Omron Sysmac Studio project UAMotionLinkLib (Sysmac Studio 1.63.0.7, LibraryProject)
(* For development of UAMotionLinkLib. *)

# Controller LIB: NX102-9000 version 1.64
Axis MC_Axis1, settings changed from default: AxisType=ServoType, FunctionLimit=SingleAxisPTP, UnitsConversion=EnumElement2, UnitsNumerator=8388608, UnitsDenominator=10, TravelDistancePerWorkRotation=5, MaxVelocity=200, MaxJogVelocity=200, InPositionBand=1, ZeroPositionBand=1, FollowingErrorLimit=5, FollowingErrorAlarmLimit=1, EncoderTypes=Abs
Axis MC_Axis2, settings changed from default: AxisNumber=1, AxisType=ServoType, FunctionLimit=SingleAxisPTP, UnitsConversion=EnumElement5, UnitsNumerator=8388608, UnitsDenominator=360, MaxVelocity=36000, MaxJogVelocity=36000, InPositionBand=0.1, ModuloMAXPosition=360, ModuloMINPosition=0
Task PrimaryTask (priority 4, period or condition 2000): ModelTest, ModelTestSimDriveReflection



PROGRAM README
RETURN;
(*

# About This Project
This project is for the development of UAMotionLinkLib.
UAMotionLinkLib provide a model FBs that control a servo via motion FBs published on an OPC UA server.
Currently, UAMotionLinkLib is intended for minor positioning operations such as trial runs and adjustments.

The model FBs are limited to providing wrappers for motion FBs related to positioning.
Servo operation preparation, stop, and emergency stop operations are provided appropriately in the user software,
and it is assumed that these are operating at an appropriate level when using UAMotionLinkLib.


# このプロジェクトについて
このプロジェクトは、UAMotionLinkLibの開発用プロジェクトです。
UAMotionLinkLibは、OPC UAサーバで公開するモーションFBを介してサーボを操作するモデルFBを提供します。
現在、UAMotionLinkLibは、試運転や調整の軽微な位置決め操作を対象としています。

モデルFBは、位置決めに関連したモーションFBのラッパー提供に限ります。
サーボ動作準備、停止、非常停止操作はユーザーソフトウェアにおいて適切に提供され、
UAMotionLinkLib使用時は、それらが適切な水準で動作していることを前提にしています。


For the parts to which I have rights, I follow POU/PROGRAM/LICENSE.
You are free to use and modify it, but we are not responsible for any damage or loss related to it.
*)
END_PROGRAM

PROGRAM LICENSE
RETURN;
(*
The MIT License (MIT)

Copyright(c) 2025 KITA Munemitsu

Permission is hereby granted, free of charge, to any person obtaining a copy of this software and associated
documentation files (the “Software”), to deal in the Software without restriction, including without limitation
the rights to use, copy, modify, merge, publish, distribute, sublicense, and/or sell copies of the Software,
and to permit persons to whom the Software is furnished to do so, subject to the following conditions:

The above copyright notice and this permission notice shall be included in all copies or substantial portions of the Software.

THE SOFTWARE IS PROVIDED “AS IS”, WITHOUT WARRANTY OF ANY KIND, EXPRESS OR IMPLIED, INCLUDING BUT NOT
LIMITED TO THE WARRANTIES OF MERCHANTABILITY, FITNESS FOR A PARTICULAR PURPOSE AND NONINFRINGEMENT.
IN NO EVENT SHALL THE AUTHORS OR COPYRIGHT HOLDERS BE LIABLE FOR ANY CLAIM, DAMAGES OR OTHER LIABILITY,
WHETHER IN AN ACTION OF CONTRACT, TORT OR OTHERWISE, ARISING FROM, OUT OF OR IN CONNECTION WITH THE SOFTWARE
OR THE USE OR OTHER DEALINGS IN THE SOFTWARE.
*)
END_PROGRAM

PROGRAM ModelTest
VAR
    BasicMCController : ModelTest_BasicMCControllerModel;
END_VAR
(*
# About This POU
This is the teesting the information model of UAMotionLinkLib.
Set up an OPC UA server and test that it can be operated by a repository client.

## Usage Steps
1. Prepare Pester for use
   Refer to the following for setup.

   "Installation and Update", Pester, https://pester.dev/docs/introduction/installation

2. Configure the Simulator's OPC UA Server
   Refer to the following for configuring the OPC UA server.

   "OPC UA User's Manual", OMRON Corporation, https://www.fa.omron.co.jp/data_pdf/mnu/w588-e1-15_nj501_nx.pdf?id=3705
   "PwshOpcUaClient", https://github.com/kmu2030/PwshOpcUaClient

   The user and password to register on the OPC UA server are as follows:

   Username: taker
   Password: chocolatepancakes

3. Run the test
   Run the following in the root directory of the cloned repository:

   ```powershell
   Invoke-Pester
   ```


# このPOUについて
UAMotionLinkLibの情報モデルのテスト。
OPC UAサーバを設定し、リポジトリのクライアントで操作できることをテストする。

## 使用手順
1. Pesterを使える状態にする
   以下を参考にセットアップする。
  
  "Installation and Update", Pester, https://pester.dev/docs/introduction/installation

2. シミュレータのOPC UAサーバを設定
   以下を参考にOPC UAサーバを設定する。
  
   "OPC UA User's Manual", OMRON Corporation, https://www.fa.omron.co.jp/data_pdf/mnu/w588-e1-15_nj501_nx.pdf?id=3705
   "PwshOpcUaClient", https://github.com/kmu2030/PwshOpcUaClient

   OPC UAサーバに登録するユーザーとパスワードは以下。

   Username: taker
   Password: chocolatepancakes

3. テストを実行
   以下をリポジトリのクローンのルートディレクトリで実行する。
  
   ```powershell
   Invoke-Pester
   ```

(c) 2025 KITA Munemitsu

*)

IF P_First_Run THEN
	BasicMCController.Enable := TRUE;
END_IF;

BasicMCController();
END_PROGRAM

PROGRAM ModelTestSimDriveReflection
VAR
    iSimMCRefrectors : ARRAY[0..15] OF SimMCReflector;
    i : UINT;
END_VAR
VAR_EXTERNAL CONSTANT
    _MC_AX : ARRAY[0..15] OF _sAXIS_REF;
END_VAR
(*

Reflects the axis command value to the current value when testing the information model of UAMotionLinkLib.


UAMotionLinkLibの情報モデルのテスト時に軸指令値を現在値に反映する。

(c) 2025 KITA Munemitsu

*)

FOR i := 0 TO 15 DO
	iSimMCRefrectors[i](Enable:=TRUE,
						Axis:=_MC_AX[i]);
END_FOR;
END_PROGRAM

FUNCTION_BLOCK BasicMCControllerModel
(* Model FB that provides motion control. *)
VAR
    MoveAbsolute : BasicMCControllerModel_moveAbsolute;
    MoveRelative : BasicMCControllerModel_moveRelative;
    MoveZeroPosition : BasicMCControllerModel_moveZeroPosition;
    Home : BasicMCControllerModel_home;
    SetPosition : BasicMCControllerModel_setPosition;
    Reset : BasicMCControllerModel_reset;
    SetAxisIndex : BasicMCControllerModel_setAxisIndex;
    AxisIndex : UINT := 0;
    Axis : _sAXIS_REF;
END_VAR
VAR_INPUT
    Enable : BOOL;
END_VAR
VAR_IN_OUT CONSTANT
    Axes : ARRAY[*] OF _sAXIS_REF;
END_VAR
VAR_INPUT
    AllowControl : BOOL := False;
END_VAR
VAR_OUTPUT
    Busy : BOOL;
END_VAR
(*

Model FB that provides motion control.


モーション操作を提供するモデルFB。

(c) 2025 KITA Munemitsu

*)

IF Enable <> Busy OR NOT AllowControl THEN
	MoveAbsolute.Execute := FALSE;
	MoveRelative.Execute := FALSE;
	MoveZeroPosition.Execute := FALSE;
	Home.Execute := FALSE;
	SetPosition.Execute := FALSE;
	Reset.Execute := FALSE;
	SetAxisIndex.Execute := FALSE;
	AxisIndex := 0;
END_IF;

Axis := Axes[AxisIndex];

MoveAbsolute(Axis:=Axes[AxisIndex]);
MoveRelative(Axis:=Axes[AxisIndex]);
MoveZeroPosition(Axis:=Axes[AxisIndex]);
Home(Axis:=Axes[AxisIndex]);
SetPosition(Axis:=Axes[AxisIndex]);
Reset(Axis:=Axes[AxisIndex]);
SetAxisIndex(Axes:=Axes, AxisIndex:=AxisIndex);

Busy := Enable
	OR MoveAbsolute.Busy
	OR MoveRelative.Busy
	OR MoveZeroPosition.Busy
	OR Home.Busy
	OR SetPosition.Busy
	OR Reset.Busy;
	
END_FUNCTION_BLOCK

FUNCTION_BLOCK BasicMCControllerModel_setAxisIndex
(* Method FB that specifies the axis to be operated. / This FB is for BasicMCController only. *)
VAR_INPUT
    Execute : BOOL;
END_VAR
VAR_IN_OUT CONSTANT
    Axes : ARRAY[*] OF _sAXIS_REF;
END_VAR
VAR_IN_OUT
    AxisIndex : UINT;
END_VAR
VAR_INPUT
    NewValue : UINT := 0;
END_VAR
VAR_OUTPUT
    Ok : BOOL;
    Done : BOOL;
END_VAR
(*

Method FB that specifies the axis to be operated.
This FB is for BasicMCController only.


操作対象とする軸を指定するメソッドFB。
このFBは、BasicMCController専用。

(c) 2025 KITA Munemitsu

*)

IF NOT Execute THEN
	IF Done THEN
		Ok := FALSE;
		Done := FALSE;
	END_IF;
	
	RETURN;
END_IF;

IF Execute AND NOT Done THEN
	Ok := NewValue < SizeOfAry(Axes);
	IF Ok THEN 
		AxisIndex := NewValue;
	END_IF;
	
	Done := TRUE;
END_IF;
END_FUNCTION_BLOCK

FUNCTION_BLOCK BasicMCControllerModel_moveAbsolute
(* Method FB that is a wrapper for MC_MoveAbsolute. / This FB is for BasicMCController only. *)
VAR
    iMC_MoveAbsolute : MC_MoveAbsolute;
    iState : UINT := 1001;
    iDirection : _eMC_DIRECTION;
    iBufferMode : _eMC_BUFFER_MODE;
END_VAR
VAR_IN_OUT CONSTANT
    Axis : _sAXIS_REF;
END_VAR
VAR_INPUT
    Position : LREAL := 0.0;
    Velocity : LREAL := 0.0;
    Acceleration : LREAL := 0.0;
    Deceleration : LREAL := 0.0;
    Jerk : LREAL := 0.0;
    Direction : UDINT := 0;
    BufferMode : UDINT := 0;
END_VAR
VAR_OUTPUT
    Busy : BOOL;
    Active : BOOL;
    Done : BOOL;
    CommandAborted : BOOL;
    Error : BOOL;
    ErrorID : WORD;
END_VAR
VAR_INPUT
    Execute : BOOL;
END_VAR
(*

Method FB that is a wrapper for MC_MoveAbsolute.
This FB is for BasicMCController only.


MC_MoveAbsoluteのラッパーであるメソッドFB。
このFBは、BasicMCController専用。

(c) 2025 KITA Munemitsu

*)

IF NOT Execute THEN
	IF iState > 0 THEN
		Error := FALSE;
		ErrorID := 0;
		CommandAborted := FALSE;
		Active := FALSE;
		Busy := FALSE;
		Done := FALSE;
		iState := 1001;
		iMC_MoveAbsolute.Execute := FALSE;
	END_IF;
ELSIF Execute AND NOT (Busy OR Done) THEN
	iState := 0;
END_IF;

CASE iState OF
	0:
		iMC_MoveAbsolute.Acceleration := Acceleration;
		iMC_MoveAbsolute.Deceleration := Deceleration;
		iMC_MoveAbsolute.Jerk := Jerk;
		iMC_MoveAbsolute.Position := Position;
		iMC_MoveAbsolute.Velocity := Velocity;
		NumToEnum(In:=Direction, InOut:=iDirection);
		iMC_MoveAbsolute.Direction := iDirection;
		NumToEnum(In:=BufferMode, InOut:=iBufferMode);
		iMC_MoveAbsolute.BufferMode := iBufferMode;
		iMC_MoveAbsolute.Execute := TRUE;
		
		Inc(iState);
	1:
		IF iMC_MoveAbsolute.Done
			OR iMC_MoveAbsolute.Error
			OR iMC_MoveAbsolute.CommandAborted
		THEN
			iMC_MoveAbsolute.Execute := FALSE;
			IF iMC_MoveAbsolute.Error THEN
				Error := TRUE;
				ErrorID := iMC_MoveAbsolute.ErrorID;
			END_IF;
			CommandAborted := iMC_MoveAbsolute.CommandAborted;
			
			Inc(iState);
		END_IF;
	2:
		IF NOT iMC_MoveAbsolute.Busy THEN
			iState := 1000;
		END_IF;
	1000:
		Done := TRUE;

		Inc(iState);
END_CASE;
Busy := iState < 1001;

iMC_MoveAbsolute(Axis:=Axis);
Active := iMC_MoveAbsolute.Active;
END_FUNCTION_BLOCK

FUNCTION_BLOCK BasicMCControllerModel_moveRelative
(* Method FB that is a wrapper for MC_MoveRelative. / This FB is for BasicMCController only. *)
VAR
    iMC_MoveRelative : MC_MoveRelative;
    iState : UINT := 1001;
    iBufferMode : _eMC_BUFFER_MODE;
END_VAR
VAR_INPUT
    Execute : BOOL;
END_VAR
VAR_IN_OUT CONSTANT
    Axis : _sAXIS_REF;
END_VAR
VAR_INPUT
    Distance : LREAL := 0.0;
    Velocity : LREAL := 0.0;
    Acceleration : LREAL := 0.0;
    Deceleration : LREAL := 0.0;
    Jerk : LREAL := 0.0;
    BufferMode : UDINT := 0;
END_VAR
VAR_OUTPUT
    Busy : BOOL;
    Active : BOOL;
    Done : BOOL;
    CommandAborted : BOOL;
    Error : BOOL;
    ErrorID : WORD;
END_VAR
(*

Method FB that is a wrapper for MC_MoveRelative.
This FB is for BasicMCController only.


MC_MoveRelativeのラッパーであるメソッドFB。
このFBは、BasicMCController専用。

(c) 2025 KITA Munemitsu

*)

IF NOT Execute THEN
	IF iState > 0 THEN
		Error := FALSE;
		ErrorID := 0;
		CommandAborted := FALSE;
		Active := FALSE;
		Busy := FALSE;
		Done := FALSE;
		iState := 1001;
		iMC_MoveRelative.Execute := FALSE;
	END_IF;
ELSIF Execute AND NOT (Busy OR Done) THEN
	iState := 0;
END_IF;

CASE iState OF
	0:
		iMC_MoveRelative.Acceleration := Acceleration;
		iMC_MoveRelative.Deceleration := Deceleration;
		iMC_MoveRelative.Jerk := Jerk;
		iMC_MoveRelative.Distance := Distance;
		iMC_MoveRelative.Velocity := Velocity;
		NumToEnum(In:=BufferMode, InOut:=iBufferMode);
		iMC_MoveRelative.BufferMode := iBufferMode;
		iMC_MoveRelative.Execute := TRUE;
		
		Inc(iState);
	1:
		IF iMC_MoveRelative.Done
			OR iMC_MoveRelative.Error
			OR iMC_MoveRelative.CommandAborted
		THEN
			iMC_MoveRelative.Execute := FALSE;
			IF iMC_MoveRelative.Error THEN
				Error := TRUE;
				ErrorID := iMC_MoveRelative.ErrorID;
			END_IF;
			CommandAborted := iMC_MoveRelative.CommandAborted;
			
			Inc(iState);
		END_IF;
	2:
		IF NOT iMC_MoveRelative.Busy THEN
			iState := 1000;
		END_IF;
	1000:
		Done := TRUE;

		Inc(iState);
END_CASE;
Busy := iState < 1001;

iMC_MoveRelative(Axis:=Axis);
Active := iMC_MoveRelative.Active;
END_FUNCTION_BLOCK

FUNCTION_BLOCK BasicMCControllerModel_moveZeroPosition
(* Method FB that is a wrapper for MC_MoveZeroPosition. / This FB is for BasicMCController only. *)
VAR
    iMC_MoveZeroPosition : MC_MoveZeroPosition;
    iState : UINT := 1001;
    iBufferMode : _eMC_BUFFER_MODE;
END_VAR
VAR_INPUT
    Execute : BOOL;
END_VAR
VAR_IN_OUT CONSTANT
    Axis : _sAXIS_REF;
END_VAR
VAR_INPUT
    Velocity : LREAL := 0.0;
    Acceleration : LREAL := 0.0;
    Deceleration : LREAL := 0.0;
    Jerk : LREAL := 0.0;
    BufferMode : UDINT := 0;
END_VAR
VAR_OUTPUT
    Busy : BOOL;
    Active : BOOL;
    Done : BOOL;
    CommandAborted : BOOL;
    Error : BOOL;
    ErrorID : WORD;
END_VAR
(*

Method FB that is a wrapper for MC_MoveZeroPosition.
This FB is for BasicMCController only.


MC_MoveZeroPositionのラッパーであるメソッドFB。
このFBは、BasicMCController専用。

(c) 2025 KITA Munemitsu

*)

IF NOT Execute THEN
	IF iState > 0 THEN
		Error := FALSE;
		ErrorID := 0;
		CommandAborted := FALSE;
		Active := FALSE;
		Busy := FALSE;
		Done := FALSE;
		iState := 1001;
		iMC_MoveZeroPosition.Execute := FALSE;
	END_IF;
ELSIF Execute AND NOT (Busy OR Done) THEN
	iState := 0;
END_IF;

CASE iState OF
	0:
		iMC_MoveZeroPosition.Acceleration := Acceleration;
		iMC_MoveZeroPosition.Deceleration := Deceleration;
		iMC_MoveZeroPosition.Jerk := Jerk;
		iMC_MoveZeroPosition.Velocity := Velocity;
		NumToEnum(In:=BufferMode, InOut:=iBufferMode);
		iMC_MoveZeroPosition.BufferMode := iBufferMode;
		iMC_MoveZeroPosition.Execute := TRUE;
		
		Inc(iState);
	1:
		IF iMC_MoveZeroPosition.Done
			OR iMC_MoveZeroPosition.Error
			OR iMC_MoveZeroPosition.CommandAborted
		THEN
			iMC_MoveZeroPosition.Execute := FALSE;
			IF iMC_MoveZeroPosition.Error THEN
				Error := TRUE;
				ErrorID := iMC_MoveZeroPosition.ErrorID;
			END_IF;
			CommandAborted := iMC_MoveZeroPosition.CommandAborted;
			
			Inc(iState);
		END_IF;
	2:
		IF NOT iMC_MoveZeroPosition.Busy THEN
			iState := 1000;
		END_IF;
	1000:
		Done := TRUE;

		Inc(iState);
END_CASE;
Busy := iState < 1001;

iMC_MoveZeroPosition(Axis:=Axis);
Active := iMC_MoveZeroPosition.Active;
END_FUNCTION_BLOCK

FUNCTION_BLOCK BasicMCControllerModel_home
(* Method FB that is a wrapper for MC_Home. / This FB is for BasicMCController only. *)
VAR
    iMC_Home : MC_Home;
    iState : UINT := 1001;
END_VAR
VAR_INPUT
    Execute : BOOL;
END_VAR
VAR_IN_OUT CONSTANT
    Axis : _sAXIS_REF;
END_VAR
VAR_OUTPUT
    Busy : BOOL;
    Done : BOOL;
    CommandAborted : BOOL;
    Error : BOOL;
    ErrorID : WORD;
END_VAR
(*

Method FB that is a wrapper for MC_Home.
This FB is for BasicMCController only.


MC_HomeのラッパーであるメソッドFB。
このFBは、BasicMCController専用。

(c) 2025 KITA Munemitsu

*)

IF NOT Execute THEN
	IF iState > 0 THEN
		Error := FALSE;
		ErrorID := 0;
		CommandAborted := FALSE;
		Busy := FALSE;
		Done := FALSE;
		iState := 1001;
		iMC_Home.Execute := FALSE;
	END_IF;
ELSIF Execute AND NOT (Busy OR Done) THEN
	iState := 0;
END_IF;

CASE iState OF
	0:
		iMC_Home.Execute := TRUE;
		
		Inc(iState);
	1:
		IF iMC_Home.Done
			OR iMC_Home.Error
			OR iMC_Home.CommandAborted
		THEN
			iMC_Home.Execute := FALSE;
			IF iMC_Home.Error THEN
				Error := TRUE;
				ErrorID := iMC_Home.ErrorID;
			END_IF;
			CommandAborted := iMC_Home.CommandAborted;
			
			Inc(iState);
		END_IF;
	2:
		IF NOT iMC_Home.Busy THEN
			iState := 1000;
		END_IF;
	1000:
		Done := TRUE;

		Inc(iState);
END_CASE;
Busy := iState < 1001;

iMC_Home(Axis:=Axis);
END_FUNCTION_BLOCK

FUNCTION_BLOCK BasicMCControllerModel_setPosition
(* Method FB that is a wrapper for MC_SetPosition. / This FB is for BasicMCController only. *)
VAR
    iMC_SetPosition : MC_SetPosition;
    iState : UINT := 1001;
    iReferenceType : _eMC_REFERENCE_TYPE;
END_VAR
VAR_INPUT
    Execute : BOOL;
END_VAR
VAR_IN_OUT CONSTANT
    Axis : _sAXIS_REF;
END_VAR
VAR_INPUT
    Position : LREAL;
    ReferenceType : UDINT;
END_VAR
VAR_OUTPUT
    Busy : BOOL;
    Done : BOOL;
    CommandAborted : BOOL;
    Error : BOOL;
    ErrorID : WORD;
END_VAR
(*

Method FB that is a wrapper for MC_SetPosition.
This FB is for BasicMCController only.


MC_SetPositionのラッパーであるメソッドFB。
このFBは、BasicMCController専用。

(c) 2025 KITA Munemitsu

*)

IF NOT Execute THEN
	IF iState > 0 THEN
		Error := FALSE;
		ErrorID := 0;
		CommandAborted := FALSE;
		Busy := FALSE;
		Done := FALSE;
		iState := 1001;
		iMC_SetPosition.Execute := FALSE;
	END_IF;
ELSIF Execute AND NOT (Busy OR Done) THEN
	iState := 0;
END_IF;

CASE iState OF
	0:
		iMC_SetPosition.Position := Position;
		NumToEnum(In:=ReferenceType, InOut:=iReferenceType);
		iMC_SetPosition.ReferenceType := iReferenceType;
	
		iMC_SetPosition.Execute := TRUE;
		
		Inc(iState);
	1:
		IF iMC_SetPosition.Done
			OR iMC_SetPosition.Error 
			OR iMC_SetPosition.CommandAborted
		THEN
			iMC_SetPosition.Execute := FALSE;
			IF iMC_SetPosition.Error THEN
				Error := TRUE;
				ErrorID := iMC_SetPosition.ErrorID;
			END_IF;
			CommandAborted := iMC_SetPosition.CommandAborted;
			
			Inc(iState);
		END_IF;
	2:
		IF NOT iMC_SetPosition.Busy THEN
			iState := 1000;
		END_IF;
	1000:
		Done := TRUE;

		Inc(iState);
END_CASE;
Busy := iState < 1001;

iMC_SetPosition(Axis:=Axis);
END_FUNCTION_BLOCK

FUNCTION_BLOCK BasicMCControllerModel_reset
(* Method FB that is a wrapper for MC_Reset. / This FB is for BasicMCController only. *)
VAR
    iMC_Reset : MC_Reset;
    iState : UINT := 1001;
END_VAR
VAR_INPUT
    Execute : BOOL;
END_VAR
VAR_IN_OUT CONSTANT
    Axis : _sAXIS_REF;
END_VAR
VAR_OUTPUT
    Busy : BOOL;
    Done : BOOL;
    Failure : BOOL;
    Error : BOOL;
    ErrorID : WORD;
END_VAR
(*

Method FB that is a wrapper for MC_Reset.
This FB is for BasicMCController only.


MC_ResetのラッパーであるメソッドFB。
このFBは、BasicMCController専用。

(c) 2025 KITA Munemitsu

*)

IF NOT Execute THEN
	IF iState > 0 THEN
		Error := FALSE;
		ErrorID := 0;
		Failure := FALSE;
		Busy := FALSE;
		Done := FALSE;
		iState := 1001;
		iMC_Reset.Execute := FALSE;
	END_IF;
ELSIF Execute AND NOT (Busy OR Done) THEN
	iState := 0;
END_IF;

CASE iState OF
	0:
		iMC_Reset.Execute := TRUE;
		
		Inc(iState);
	1:
		IF iMC_Reset.Done
			OR iMC_Reset.Error
			OR iMC_Reset.Failure
		THEN
			iMC_Reset.Execute := FALSE;
			IF iMC_Reset.Error THEN
				Error := TRUE;
				ErrorID := iMC_Reset.ErrorID;
			END_IF;
			Failure := iMC_Reset.Failure;
			
			Inc(iState);
		END_IF;
	2:
		IF NOT iMC_Reset.Busy THEN
			iState := 1000;
		END_IF;
	1000:
		Done := TRUE;

		Inc(iState);
END_CASE;
Busy := iState < 1001;

iMC_Reset(Axis:=Axis);
END_FUNCTION_BLOCK

FUNCTION_BLOCK ModelTest_BasicMCControllerModel
(* Public FB for the test controller of BasicMCControllerModel. *)
VAR
    Target : BasicMCControllerModel;
    iResetMCError : ResetMCError;
    iMC_Power : MC_Power;
    iMC_Stop : MC_Stop;
    iMC_Home : MC_Home;
    iSIM_SetDrvAlm : SIM_SetDrvAlm;
    iSIM_SetDrvWarn : SIM_SetDrvWarn;
    iSIM_SigEmergeStop : SIM_SigEmergStop;
    iSIM_SigPosLmt : SIM_SigPosLmt;
    iSIM_SigNegLmt : SIM_SigNegLmt;
    Initialize : ModelTest_stateMethod;
    InitializeCount : UINT := 0;
    iInitializeContext : UINT := 0;
    ServoOn : ModelTest_stateMethod;
    ServoOnCount : UINT := 0;
    iServoOnContext : UINT := 0;
    ServoOff : ModelTest_stateMethod;
    ServoOffCount : UINT := 0;
    iServoOffContext : UINT := 0;
    Stop : ModelTest_stateMethod;
    StopCount : UINT := 0;
    iStopContext : UINT := 0;
    Home : ModelTest_stateMethod;
    HomeCount : UINT := 0;
    iHomeContext : UINT := 0;
    SetAxisIndex : ModelTest_stateMethodWithUintArg;
    SetAxisIndexCount : UINT := 0;
    iSetAxisIndexContext : UINT := 0;
    FireDriverAlarm : ModelTest_stateMethod;
    FireDriverAlarmCount : UINT := 0;
    iFireDriverAlarmContext : UINT := 0;
    FireDriverWarning : ModelTest_stateMethod;
    FireDriverWarningCount : UINT := 0;
    iFireDriverWarningContext : UINT := 0;
    FirePositiveLimitSignal : ModelTest_stateEnableMethod;
    FirePositiveLimitSignalCount : UINT := 0;
    iFirePositiveLimitSignalContext : UINT := 0;
    FireNegativeLimitSignal : ModelTest_stateEnableMethod;
    FireNegativeLimitSignalCount : UINT := 0;
    iFireNegativeLimitSignalContext : UINT := 0;
    FireEmergencyStopSignal : ModelTest_stateEnableMethod;
    FireEmergencyStopSignalCount : UINT := 0;
    iFireEmergencyStopSignalContext : UINT := 0;
    TearDown : ModelTest_stateMethod;
    TearDownCount : UINT := 0;
    iTearDownContext : UINT := 0;
    AxisIndex : UINT := 0;
END_VAR
VAR_INPUT
    Enable : BOOL;
END_VAR
VAR_OUTPUT
    Busy : BOOL;
END_VAR
VAR_EXTERNAL CONSTANT
    _MC_AX : ARRAY[0..15] OF _sAXIS_REF;
END_VAR
(*

Public FB for the test controller of BasicMCControllerModel.


BasicMCControllerModelのテストコントローラ公開FB。

(c) 2025 KITA Munemitsu

*)

IF Enable AND NOT Busy THEN
	Initialize.Execute := FALSE;
	Clear(iInitializeContext);
	Clear(InitializeCount);

	ServoOn.Execute := FALSE;
	Clear(iServoOnContext);
	Clear(ServoOnCount);

	ServoOff.Execute := FALSE;
	Clear(iServoOffContext);
	Clear(ServoOffCount);

	Stop.Execute := FALSE;
	Clear(iStopContext);
	Clear(StopCount);

	Home.Execute := FALSE;
	Clear(iHomeContext);
	Clear(HomeCount);

	SetAxisIndex.Execute := FALSE;
	Clear(iSetAxisIndexContext);
	Clear(SetAxisIndexCount);

	FireDriverAlarm.Execute := FALSE;
	Clear(iFireDriverAlarmContext);
	Clear(FireDriverAlarmCount);

	FireDriverAlarm.Execute := FALSE;
	Clear(iFireDriverAlarmContext);
	Clear(FireDriverAlarmCount);

	FirePositiveLimitSignal.Enable := FALSE;
	Clear(iFirePositiveLimitSignalContext);
	Clear(FirePositiveLimitSignalCount);

	FireNegativeLimitSignal.Enable := FALSE;
	Clear(iFireNegativeLimitSignalContext);
	Clear(FireNegativeLimitSignalCount);

	FireEmergencyStopSignal.Enable := FALSE;
	Clear(iFireEmergencyStopSignalContext);
	Clear(FireEmergencyStopSignalCount);

	TearDown.Execute := FALSE;
	Clear(iTearDownContext);
	Clear(TearDownCount);
	
	Target.AllowControl := TRUE;
	Target.Enable := TRUE;
		
	Busy := TRUE;
ELSIF NOT Enable AND Busy THEN
	Initialize.Execute := FALSE;
	ServoOn.Execute := FALSE;
	ServoOff.Execute := FALSE;
	Stop.Execute := FALSE;
	Home.Execute := FALSE;
	SetAxisIndex.Execute := FALSE;
	FireDriverAlarm.Execute := FALSE;
	FireDriverWarning.Execute := FALSE;
	FirePositiveLimitSignal.Enable := FALSE;
	FireNegativeLimitSignal.Enable := FALSE;
	FireEmergencyStopSignal.Enable := FALSE;
	TearDown.Execute := FALSE;
	
	Target.Enable := FALSE;
	
	Busy := FALSE;	
END_IF;

IF Busy THEN
	Initialize(Context:=iInitializeContext);
	IF Initialize.Busy THEN
		CASE iInitializeContext OF
			// Init
			0:
				iMC_Power.Enable := FALSE;
				Target.Enable := FALSE;
				
				Inc(iInitializeContext);
			1:
				IF GetMCError() THEN
					iResetMCError.Execute := TRUE;
					
					Inc(iInitializeContext);
				ELSE
					iInitializeContext := iInitializeContext + 2;
				END_IF;
			2:
				IF iResetMCError.Done OR iResetMCError.Error THEN
					iResetMCError.Execute := FALSE;
					
					Inc(iInitializeContext);
				END_IF;
			3:
				Target.Enable := TRUE;
				
				iInitializeContext := 1000;
				
			// Done
			1000:
				Inc(InitializeCount);
				
				Inc(iInitializeContext);
		END_CASE;
	END_IF;

	ServoOn(Context:=iServoOnContext);
	IF ServoOn.Busy THEN
		CASE iServoOnContext OF
			// Init
			0:
				iMC_Power.Enable := TRUE;
				
				Inc(iServoOnContext);
			1:
				IF iMC_Power.Busy THEN
					iServoOnContext := 1000;
				END_IF;
			
			// Done
			1000:
				Inc(ServoOnCount);
			
				Inc(iServoOnContext);
		END_CASE;
	END_IF;

	ServoOff(Context:=iServoOffContext);
	IF ServoOff.Busy THEN
		CASE iServoOffContext OF
			// Init
			0:
				iMC_Power.Enable := FALSE;
				
				Inc(iServoOffContext);
			1:
				IF NOT iMC_Power.Busy THEN
					iServoOffContext := 1000;
				END_IF;
			
			// Done
			1000:
				Inc(ServoOffCount);
			
				Inc(iServoOffContext);
		END_CASE;
	END_IF;

	Stop(Context:=iStopContext);
	IF Stop.Busy THEN
		CASE iStopContext OF
			// Init
			0:
				iMC_Stop.Execute := TRUE;
				
				Inc(iStopContext);
			1:
				IF iMC_Stop.Done OR iMC_Stop.Error THEN
					iMC_Stop.Execute := FALSE;
					
					iStopContext := 1000;
				END_IF;
			
			// Done
			1000:
				Inc(StopCount);
			
				Inc(iStopContext);
		END_CASE;
	ELSE
		iMC_Stop.Execute := FALSE;
	END_IF;

	Home(Context:=iHomeContext);
	IF Home.Busy THEN
		CASE iHomeContext OF
			// Init
			0:
				iMC_Home.Execute := TRUE;
				
				Inc(iHomeContext);
			1:
				IF iMC_Home.Done OR iMC_Home.Error THEN
					iMC_Home.Execute := FALSE;
					
					iHomeContext := 1000;
				END_IF;
			
			// Done
			1000:
				Inc(HomeCount);
			
				Inc(iHomeContext);
		END_CASE;
	ELSE
		iMC_Home.Execute := FALSE;
	END_IF;

	SetAxisIndex(Context:=iSetAxisIndexContext);
	IF SetAxisIndex.Busy THEN
		CASE iSetAxisIndexContext OF
			// Init
			0:
				AxisIndex := SetAxisIndex.Value;
				
				iSetAxisIndexContext := 1000;
			
			// Done
			1000:
				Inc(SetAxisIndexCount);
			
				Inc(iSetAxisIndexContext);
		END_CASE;
	END_IF;

	FireDriverAlarm(Context:=iFireDriverAlarmContext);
	IF FireDriverAlarm.Busy THEN
		CASE iFireDriverAlarmContext OF
			// Init
			0:
				iSIM_SetDrvAlm.Execute := TRUE;
				
				Inc(iFireDriverAlarmContext);
			1:
				IF iSIM_SetDrvAlm.Done OR iSIM_SetDrvAlm.Error THEN
					iSIM_SetDrvAlm.Execute := FALSE;
					
					iFireDriverAlarmContext := 1000;
				END_IF;

			// Done
			1000:
				Inc(FireDriverAlarmCount);
			
				Inc(iFireDriverAlarmContext);
		END_CASE;
	ELSE
		iSIM_SetDrvAlm.Execute := FALSE;
	END_IF;

	FireDriverWarning(Context:=iFireDriverWarningContext);
	IF FireDriverWarning.Busy THEN
		CASE iFireDriverWarningContext OF
			// Init
			0:
				iSIM_SetDrvWarn.Execute := TRUE;
				
				Inc(iFireDriverWarningContext);
			1:
				IF iSIM_SetDrvWarn.Done OR iSIM_SetDrvWarn.Error THEN
					iSIM_SetDrvWarn.Execute := FALSE;
					
					iFireDriverWarningContext := 1000;
				END_IF;

			// Done
			1000:
				Inc(FireDriverWarningCount);
			
				Inc(iFireDriverWarningContext);
		END_CASE;
	ELSE
		iSIM_SetDrvWarn.Execute := FALSE;
	END_IF;

	FirePositiveLimitSignal(Context:=iFirePositiveLimitSignalContext);
	IF FirePositiveLimitSignal.Busy THEN
		CASE iFirePositiveLimitSignalContext OF
			// Init
			0:
				iSIM_SigPosLmt.Enable := TRUE;
				
				Inc(iFirePositiveLimitSignalContext);
			1:
				IF iSIM_SigPosLmt.Status THEN
					iFirePositiveLimitSignalContext := 10;
				END_IF;
			
			// Active
			10:
				IF NOT FirePositiveLimitSignal.Enable THEN
					iSIM_SigPosLmt.Enable := FALSE;
					
					iFirePositiveLimitSignalContext := 1000;
				END_IF;

			// Done
			1000:
				Inc(FirePositiveLimitSignalCount);
			
				Inc(iFirePositiveLimitSignalContext);
		END_CASE;
	ELSE
		iSIM_SigPosLmt.Enable := FALSE;
	END_IF;

	FireNegativeLimitSignal(Context:=iFireNegativeLimitSignalContext);
	IF FireNegativeLimitSignal.Busy THEN
		CASE iFireNegativeLimitSignalContext OF
			// Init
			0:
				iSIM_SigNegLmt.Enable := TRUE;
				
				Inc(iFireNegativeLimitSignalContext);
			1:
				IF iSIM_SigNegLmt.Status THEN
					iFireNegativeLimitSignalContext := 10;
				END_IF;
			
			// Active
			10:
				IF NOT FireNegativeLimitSignal.Enable THEN
					iSIM_SigNegLmt.Enable := FALSE;
					
					iFireNegativeLimitSignalContext := 1000;
				END_IF;

			// Done
			1000:
				Inc(FireNegativeLimitSignalCount);
			
				Inc(iFireNegativeLimitSignalContext);
		END_CASE;
	ELSE
		iSIM_SigNegLmt.Enable := FALSE;
	END_IF;

	FireEmergencyStopSignal(Context:=iFireEmergencyStopSignalContext);
	IF FireEmergencyStopSignal.Busy THEN
		CASE iFireEmergencyStopSignalContext OF
			// Init
			0:
				iSIM_SigEmergeStop.Enable := TRUE;
				
				Inc(iFireEmergencyStopSignalContext);
			1:
				IF iSIM_SigEmergeStop.Status THEN
					iFireEmergencyStopSignalContext := 10;
				END_IF;
			
			// Active
			10:
				IF NOT FireEmergencyStopSignal.Enable THEN
					iSIM_SigEmergeStop.Enable := FALSE;
					
					iFireEmergencyStopSignalContext := 1000;
				END_IF;

			// Done
			1000:
				Inc(iFireEmergencyStopSignalContext);
			
				Inc(iFireEmergencyStopSignalContext);
		END_CASE;
	ELSE
		iSIM_SigEmergeStop.Enable := FALSE;
	END_IF;

	TearDown(Context:=iTearDownContext);
	IF TearDown.Busy THEN
		CASE iTearDownContext OF
			// Init
			0:
				iMC_Power.Enable := FALSE;
				Target.Enable := FALSE;
				
				Inc(iTearDownContext);
			1:
				IF GetMCError() THEN
					iResetMCError.Execute := TRUE;
					
					Inc(iTearDownContext);
				ELSE
					iTearDownContext := iTearDownContext + 2;
				END_IF;
			2:
				IF iResetMCError.Done OR iResetMCError.Error THEN
					iResetMCError.Execute := FALSE;
					
					Inc(iTearDownContext);
				END_IF;
			3:
				Target.Enable := TRUE;
				
				iTearDownContext := 1000;
				
			// Done
			1000:
				Inc(TearDownCount);
				
				Inc(iTearDownContext);
		END_CASE;
	END_IF;
END_IF;

iResetMCError();
iMC_Power(Axis:=_MC_AX[AxisIndex]);
iMC_Stop(Axis:=_MC_AX[AxisIndex]);
iMC_Home(Axis:=_MC_AX[AxisIndex]);

iSIM_SigPosLmt(Axis:=_MC_AX[AxisIndex]);
iSIM_SigNegLmt(Axis:=_MC_AX[AxisIndex]);
iSIM_SigEmergeStop(Axis:=_MC_AX[AxisIndex]);
iSIM_SetDrvAlm(Axis:=_MC_AX[AxisIndex]);
iSIM_SetDrvWarn(Axis:=_MC_AX[AxisIndex]);

Target(Axes:=_MC_AX);
END_FUNCTION_BLOCK

FUNCTION_BLOCK ModelTest_stateMethod
VAR_INPUT
    Execute : BOOL;
END_VAR
VAR_IN_OUT
    Context : UINT;
END_VAR
VAR_OUTPUT
    Busy : BOOL;
    Done : BOOL;
END_VAR
IF Execute AND NOT Busy THEN
	Busy := TRUE;
ELSIF NOT Execute AND Busy THEN
	Context := 0;
	Busy := FALSE;
	Done := FALSE;
ELSIF Busy THEN
	Done := Context >= 1000;
ELSIF NOT Execute THEN
	Context := 0;
	Done := FALSE;
END_IF;
END_FUNCTION_BLOCK

FUNCTION_BLOCK ModelTest_stateMethodWithUintArg
VAR_INPUT
    Execute : BOOL;
END_VAR
VAR_IN_OUT
    Context : UINT;
END_VAR
VAR_OUTPUT
    Value : UINT;
    Busy : BOOL;
    Done : BOOL;
END_VAR
IF Execute AND NOT Busy THEN
	Busy := TRUE;
ELSIF NOT Execute AND Busy THEN
	Context := 0;
	Busy := FALSE;
	Done := FALSE;
ELSIF Busy THEN
	Done := Context >= 1000;
ELSIF NOT Execute THEN
	Context := 0;
	Done := FALSE;
END_IF;
END_FUNCTION_BLOCK

FUNCTION_BLOCK ModelTest_stateEnableMethod
VAR_INPUT
    Enable : BOOL;
END_VAR
VAR_IN_OUT
    Context : UINT;
END_VAR
VAR_OUTPUT
    Busy : BOOL;
END_VAR
IF Enable AND NOT Busy THEN
	Context := 0;
	Busy := TRUE;
ELSIF Busy AND Context > 1000 THEN
	Busy := FALSE;
END_IF;
END_FUNCTION_BLOCK

FUNCTION_BLOCK SimMCReflector
VAR
    iSimSetActPos : SIM_SetActPos;
    iSimSetActVel : SIM_SetActVel;
    iSimSetActTrq : SIM_SetActTrq;
    iSimSigNegLim : SIM_SigNegLmt;
    iSimSigPosLim : SIM_SigPosLmt;
END_VAR
VAR CONSTANT
    STATE_INIT : UINT := 0;
    STATE_WAIT : UINT := 10;
    STATE_REFRECT_MOTION : UINT := 20;
    STATE_DONE : UINT := 1000;
END_VAR
VAR
    iState : UINT := 1001;
END_VAR
VAR_INPUT
    Enable : BOOL;
END_VAR
VAR_IN_OUT CONSTANT
    Axis : _sAXIS_REF;
END_VAR
VAR_OUTPUT
    Busy : BOOL;
END_VAR
(*

During simulation, the operation command value is reflected in the current value.


シミュレーション時に動作指令値を現在値に反映する。

(c) 2025 KITA Munemitsu

*)

CASE Axis.Cfg.AxEnable OF
	_eMC_AXIS_USE#_mcNoneAxis,
	_eMC_AXIS_USE#_mcUnusedAxis:
		RETURN;
END_CASE;

IF Enable AND NOT Busy THEN
	Busy := TRUE;
	
	iState := STATE_INIT;
END_IF;

CASE iState OF
	// STATE_INIT
	0:
		iSimSetActPos.Enable := FALSE;
		iSimSetActVel.Enable := FALSE;
		iSimSetActTrq.Enable := FALSE;
		
		iState := STATE_WAIT;
	
	// STATE_WAIT
	10:
		IF NOT Enable THEN
			iState := STATE_DONE;
		ELSIF NOT Axis.Status.Standstill THEN
			iSimSetActPos.SetPos := Axis.Cmd.Pos;
			iSimSetActVel.SetVel := Axis.Cmd.Vel;
			iSimSetActTrq.SetTrq := Axis.Cmd.Trq;
			iSimSetActPos.Enable := TRUE;
			iSimSetActVel.Enable := TRUE;
			iSimSetActTrq.Enable := TRUE;

			iState := STATE_REFRECT_MOTION;
		END_IF;

	// STATE_REFRECT_MOTION
	20:
		iSimSetActPos.SetPos := Axis.Cmd.Pos;
		iSimSetActVel.SetVel := Axis.Cmd.Vel;
		iSimSetActTrq.SetTrq := Axis.Cmd.Trq;
		IF Axis.Status.Standstill THEN
			iState := iState + 9;
		END_IF;
	29:
		iSimSetActPos.Enable := FALSE;
		iSimSetActVel.Enable := FALSE;
		iSimSetActTrq.Enable := FALSE;
		
		iState := STATE_WAIT;
	
	// STATE_DONE
	1000:
		iSimSetActPos.Enable := FALSE;
		iSimSetActVel.Enable := FALSE;
		iSimSetActTrq.Enable := FALSE;
		
		Busy := FALSE;
		
		Inc(iState);
END_CASE;

iSimSetActPos(Axis:=Axis);
iSimSetActVel(Axis:=Axis);
iSimSetActTrq(Axis:=Axis);
END_FUNCTION_BLOCK